FUNCTION_BLOCK FB_Conveyor 
VAR_INPUT
END_VAR
VAR_OUTPUT
END_VAR
VAR
	bStart AT%Q* : BOOL;
END_VAR

METHOD Off : BOOL
VAR_INPUT
END_VAR
END_METHOD

METHOD On : BOOL
VAR_INPUT
END_VAR
END_METHOD

END_FUNCTION_BLOCK

(* stored: Version 1.1.0.1, ProductVersion 3.1.4024.0
   POU FB_Conveyor: Id {b15311d8-a9f4-4077-9cec-ef51ff0c9999}, SpecialFunc None
   Method Off: Id {f085c888-d730-4182-bd45-298546b54d73}
   Method On: Id {5d342f49-f715-42fd-b4a3-ca7fc5d5e1e7} *)
